// Mitsubishi GX Works2 project: Retentive timer   PLC: FX1N/FX1NC

PROGRAM MAIN
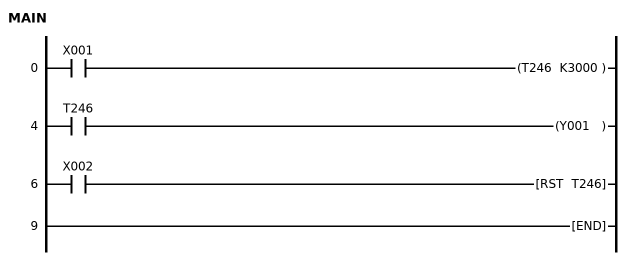
0     LD      X001
      OUT     T246 K3000
4     LD      T246
      OUT     Y001
6     LD      X002
      RST     T246
9     END
END_PROGRAM
